// Mitsubishi GX Works2 project: BookEX6_49 PID   PLC: Q13UDV

// global labels: Global
VAR_GLOBAL
  bVar0 AT M5000 : BOOL;
  abArray0 AT M5010 : ARRAY [0..49] OF BOOL;
  sStr0 AT D5000 : STRING[199];
  sStr1 AT D5100 : STRING[199];
  sStr2 AT D5200 : STRING[199];
  sStr3 AT D5300 : STRING[199];
  sStr4 AT D5400 : STRING[199];
  sStr5 AT D5500 : STRING[199];
  sStr6 AT D5600 : STRING[199];
  sStr7 AT D5700 : STRING[199];
  sStr8 AT D5800 : STRING[199];
  sStr9 AT D5900 : STRING[199];
  iVar0 AT D4500 : INT;
  iVar1 AT D4501 : INT;
  iVar2 AT D4502 : INT;
  iVar3 AT D4503 : INT;
  iVar4 AT D4504 : INT;
  iVar5 AT D4505 : INT;
  iVar6 AT D4506 : INT;
  iVar7 AT D4507 : INT;
  iVar8 AT D4508 : INT;
  iVar9 AT D4509 : INT;
  dVar0 AT D4510 : DINT;
  dVar1 AT D4512 : DINT;
  dVar2 AT D4514 : DINT;
  dVar3 AT D4516 : DINT;
  dVar4 AT D4518 : DINT;
  dVar5 AT D4520 : DINT;
  dVar6 AT D4522 : DINT;
  dVar7 AT D4524 : DINT;
  dVar8 AT D4526 : DINT;
  dVar9 AT D4528 : DINT;
  wVar0 AT D4530 : WORD;
  wVar1 AT D4531 : WORD;
  wVar2 AT D4532 : WORD;
  wVar3 AT D4533 : WORD;
  wVar4 AT D4534 : WORD;
  wVar5 AT D4535 : WORD;
  wVar6 AT D4536 : WORD;
  wVar7 AT D4537 : WORD;
  wVar8 AT D4538 : WORD;
  wVar9 AT D4539 : WORD;
  dwVar0 AT D4540 : DWORD;
  dwVar1 AT D4542 : DWORD;
  dwVar2 AT D4544 : DWORD;
  dwVar3 AT D4546 : DWORD;
  dwVar4 AT D4548 : DWORD;
  dwVar5 AT D4550 : DWORD;
  dwVar6 AT D4552 : DWORD;
  dwVar7 AT D4554 : DWORD;
  dwVar8 AT D4556 : DWORD;
  dwVar9 AT D4558 : DWORD;
  fsVar0 AT D4560 : REAL;
  fsVar1 AT D4562 : REAL;
  fsVar2 AT D4564 : REAL;
  fsVar3 AT D4566 : REAL;
  fsVar4 AT D4568 : REAL;
  fsVar5 AT D4570 : REAL;
  fsVar6 AT D4572 : REAL;
  fsVar7 AT D4574 : REAL;
  fsVar8 AT D4576 : REAL;
  fsVar9 AT D4578 : REAL;
  fdVar0 AT D4580 : LREAL;
  tTime0 AT D4620 : TIME;
  tTime1 AT D4622 : TIME;
  tTime2 AT D4624 : TIME;
  tTime3 AT D4626 : TIME;
  tTime4 AT D4628 : TIME;
  tTime5 AT D4630 : TIME;
  tTime6 AT D4632 : TIME;
  tTime7 AT D4634 : TIME;
  tTime8 AT D4636 : TIME;
  tTime9 AT D4638 : TIME;
  tTime10 AT D4640 : TIME;
  bVar1 AT M5001 : BOOL;
  bVar2 AT M5002 : BOOL;
  bVar3 AT M5003 : BOOL;
  bVar4 AT M5004 : BOOL;
  bVar5 AT M5005 : BOOL;
  bVar6 AT M5006 : BOOL;
  bVar7 AT M5007 : BOOL;
  bVar8 AT M5008 : BOOL;
  bVar9 AT M5009 : BOOL;
  abArray1 AT M5060 : ARRAY [0..49] OF BOOL;
  abArray2 AT M5110 : ARRAY [0..49] OF BOOL;
  abArray3 AT M5160 : ARRAY [0..49] OF BOOL;
  abArray4 AT M5210 : ARRAY [0..49] OF BOOL;
  abArray5 AT M5260 : ARRAY [0..49] OF BOOL;
  abArray6 AT M5310 : ARRAY [0..49] OF BOOL;
  abArray7 AT M5360 : ARRAY [0..49] OF BOOL;
  abArray8 AT M5410 : ARRAY [0..49] OF BOOL;
  abArray9 AT M5460 : ARRAY [0..49] OF BOOL;
  fdVar1 AT D4584 : LREAL;
  fdVar2 AT D4588 : LREAL;
  fdVar3 AT D4592 : LREAL;
  fdVar4 AT D4596 : LREAL;
  fdVar5 AT D4600 : LREAL;
  fdVar6 AT D4604 : LREAL;
  fdVar7 AT D4608 : LREAL;
  fdVar8 AT D4612 : LREAL;
  fdVar9 AT D4616 : LREAL;
  afsPen0 AT D2000 : ARRAY [0..499] OF REAL;
  afsPen1 AT D3000 : ARRAY [0..499] OF REAL;
END_VAR
// user libraries (not included): HMI

PROGRAM ExPIDGraph
VAR
  ix : INT;
  iy : INT;
  fsPV : REAL;
  fsEV : REAL;
  fsLastEV : REAL;
  fsIV : REAL;
  fsDV : REAL;
  fsSV : REAL;
  fsKp : REAL;
  fsKi : REAL;
  fsKd : REAL;
  fsDT : REAL;
  fsOut : REAL;
  fsLastPV : REAL;
END_VAR
;
IF SM402 THEN
	fsVar8 := -20.0;		(* Min *)
	fsVar9 := 20.0;		(* Max *)
	ix := 0;
	fsSV := 10.0;
	fsPV := 0.0;
	fsIV := 0.0;
	fsDV := 0.0;
	fsLastEV := 0.0;
	fsVar0 := 2.0;
	fsVar1 := 10.0;
	fsVar2 := 0.2;
	FOR iy:=0 TO 359 DO 
		IF iy > 300 THEN
			afsPen0[iy] := 0.0;
		ELSIF iy > 170 THEN
			afsPen0[iy] := fsSV * -1.0;
		ELSIF iy > 40 THEN
			afsPen0[iy] := fsSV;
		ELSE
			afsPen0[iy] := 0.0;
		END_IF;
	END_FOR;		
	sStr0 := 'P Gain';
	sStr1 := 'I Gain';
	sStr2 := 'D Gain';
	sStr3 := '';
	sStr4 := '';
	fsVar3 := 0.0;
	iVar4 := 0;
END_IF;

IF LDP(TRUE, SM410)  THEN 
	CASE ix OF 
		0..359 : (* PID-Control *)
					fsDT := 0.1;			
					fsEV := fsPV - afsPen0[ix];
					fsIV := fsIV + fsEV * fsDT;
					fsDV := (fsEV - fsLastEV) / fsDT;
					fsLastEV := fsEV;  
					fsOut := fsVar0 * fsEV + fsVar1 * fsIV + fsVar2 * fsDV; 
					fsPV := fsLastPV - fsOut * fsDT;
					fsLastPV := fsPV;
					(* Limit *)
					IF (fsPV > fsVar9) THEN fsPV := fsVar9;  END_IF;
					IF (fsPV < fsVar8) THEN  fsPV := fsVar8;  END_IF;
 					FOR iy:=ix TO 359 DO 
						afsPen1[iy] := fsPV;
					END_FOR;    
					ix := ix + 1;		
	ELSE
		ix := 0;
		fsPV := 0.0;
		fsIV := 0.0;
		fsDV := 0.0;
		fsLastEV := 0.0;
		FOR iy:=0 TO 359 DO 
				afsPen1[iy] := 0.0;
		END_FOR;		
	END_CASE;
END_IF;
END_PROGRAM

PROGRAM ExPID
VAR
  Mov8INT_1 : Mov8INT;
  aCtrlData : ARRAY [0..28] OF INT;
  iSV : INT;
  iPV : INT;
  iMV : INT;
  Mov8INT_2 : Mov8INT;
  Mov8INT_3 : Mov8INT;
  fsMV : REAL;
  HMI06_1 : HMI06;
END_VAR
(* structured ladder/FBD written out as ST: instructions are called as NAME(EN, inputs, outputs); _pN, _eN, _tN stand for wires *)
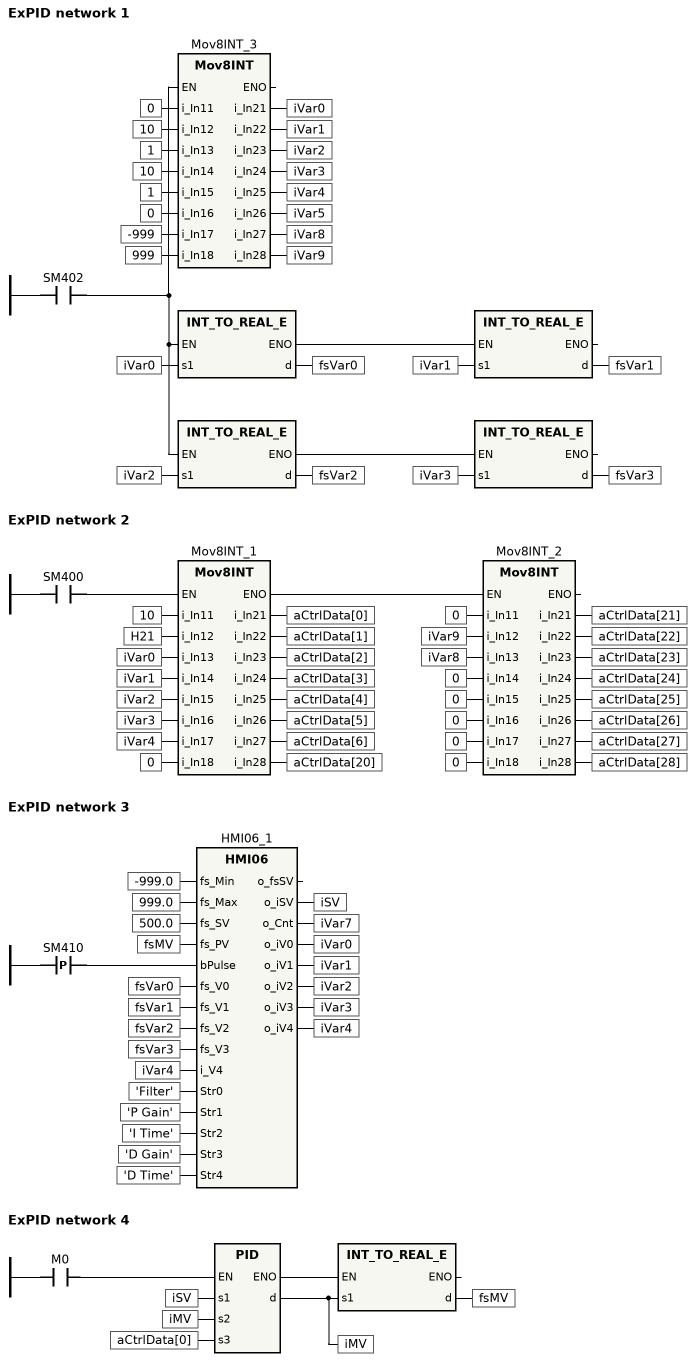
(* network 1 *)
Mov8INT_3(EN := SM402, i_In11 := 0, i_In12 := 10, i_In13 := 1, i_In14 := 10, i_In15 := 1, i_In16 := 0, i_In17 := -999, i_In18 := 999, i_In21 => iVar0, i_In22 => iVar1, i_In23 => iVar2, i_In24 => iVar3, i_In25 => iVar4, i_In26 => iVar5, i_In27 => iVar8, i_In28 => iVar9);
_e1 := INT_TO_REAL_E(SM402, iVar0, fsVar0);
INT_TO_REAL_E(_e1, iVar1, fsVar1);
_e2 := INT_TO_REAL_E(SM402, iVar2, fsVar2);
INT_TO_REAL_E(_e2, iVar3, fsVar3);
(* network 2 *)
Mov8INT_1(EN := SM400, i_In11 := 10, i_In12 := H21, i_In13 := iVar0, i_In14 := iVar1, i_In15 := iVar2, i_In16 := iVar3, i_In17 := iVar4, i_In18 := 0, i_In21 => aCtrlData[0], i_In22 => aCtrlData[1], i_In23 => aCtrlData[2], i_In24 => aCtrlData[3], i_In25 => aCtrlData[4], i_In26 => aCtrlData[5], i_In27 => aCtrlData[6], i_In28 => aCtrlData[20]);
Mov8INT_2(EN := Mov8INT_1.ENO, i_In11 := 0, i_In12 := iVar9, i_In13 := iVar8, i_In14 := 0, i_In15 := 0, i_In16 := 0, i_In17 := 0, i_In18 := 0, i_In21 => aCtrlData[21], i_In22 => aCtrlData[22], i_In23 => aCtrlData[23], i_In24 => aCtrlData[24], i_In25 => aCtrlData[25], i_In26 => aCtrlData[26], i_In27 => aCtrlData[27], i_In28 => aCtrlData[28]);
(* network 3 *)
HMI06_1(fs_Min := -999.0, fs_Max := 999.0, fs_SV := 500.0, fs_PV := fsMV, bPulse := LDP(TRUE, SM410), fs_V0 := fsVar0, fs_V1 := fsVar1, fs_V2 := fsVar2, fs_V3 := fsVar3, i_V4 := iVar4, Str0 := 'Filter', Str1 := 'P Gain', Str2 := 'I Time', Str3 := 'D Gain', Str4 := 'D Time', o_iSV => iSV, o_Cnt => iVar7, o_iV0 => iVar0, o_iV1 => iVar1, o_iV2 => iVar2, o_iV3 => iVar3, o_iV4 => iVar4);
(* network 4 *)
_e1 := PID(M0, iSV, iMV, aCtrlData[0], iMV);
INT_TO_REAL_E(_e1, iMV, fsMV);
END_PROGRAM

PROGRAM ExInexactPRMW
VAR
  Mov8INT_1 : Mov8INT;
  Mov8INT_2 : Mov8INT;
  aCtrlData : ARRAY [0..99] OF INT;
  aCtrlCont : ARRAY [0..172] OF INT;
  Mov4INT_1 : Mov4INT;
  HMI06_1 : HMI06;
  iMV : INT;
  fsMV : REAL;
  Mov8INT_3 : Mov8INT;
  fsSV : REAL;
  iSV : INT;
  Mov8INT_4 : Mov8INT;
  Mov8INT_5 : Mov8INT;
  Mov4INT_2 : Mov4INT;
  aPrmwData : ARRAY [0..99] OF INT;
END_VAR
(* structured ladder/FBD written out as ST: instructions are called as NAME(EN, inputs, outputs); _pN, _eN, _tN stand for wires *)
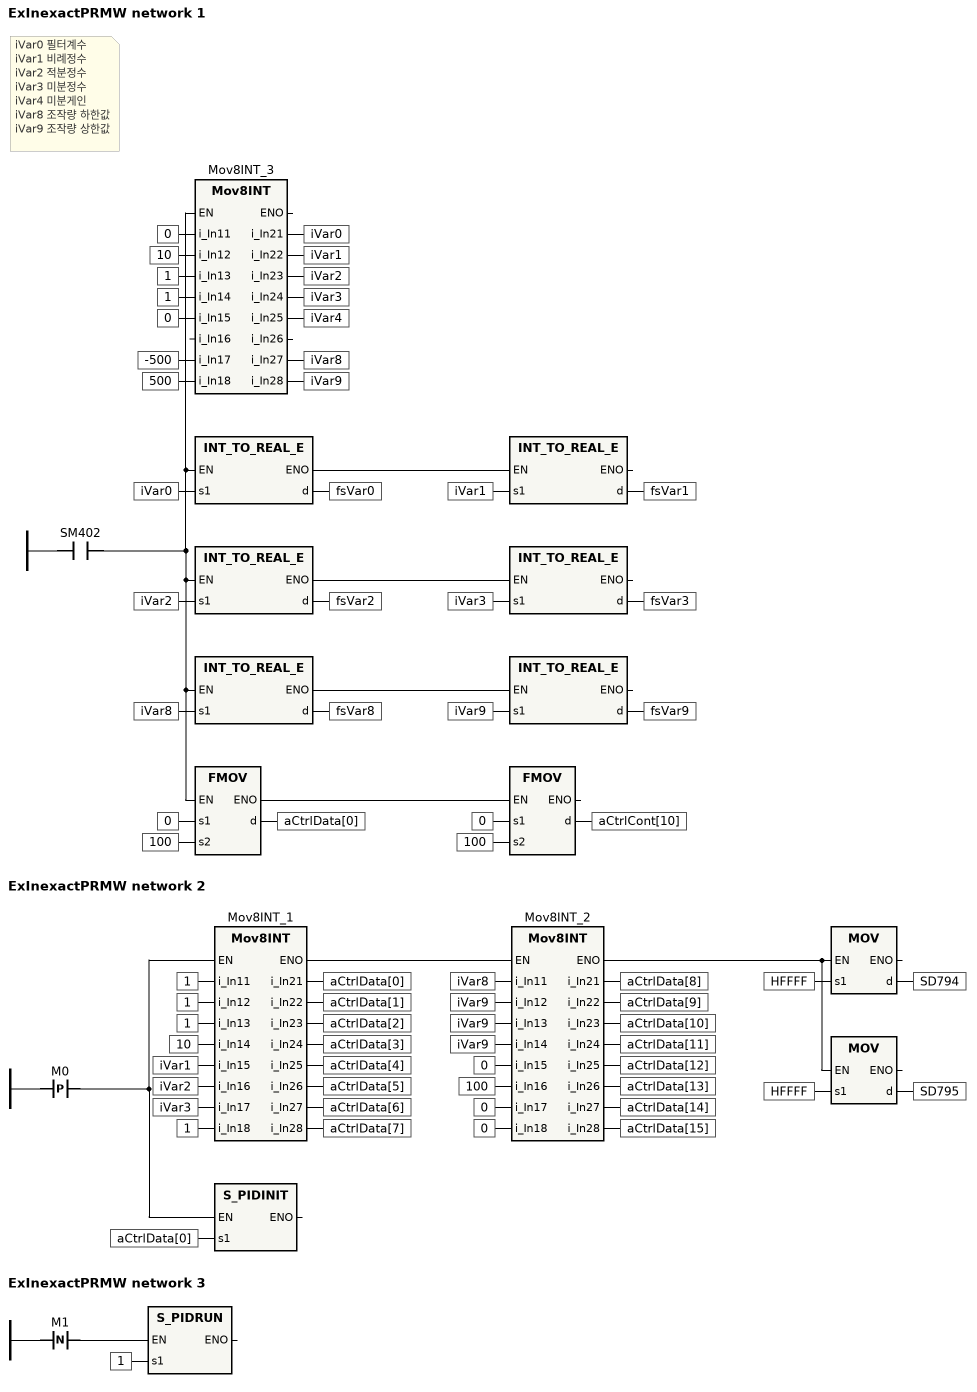
(* network 1 *)
(* iVar0 필터계수 / iVar1 비례정수 / iVar2 적분정수 / iVar3 미분정수 / iVar4 미분게인 / iVar8 조작량 하한값 / iVar9 조작량 상한값 *)
Mov8INT_3(EN := SM402, i_In11 := 0, i_In12 := 10, i_In13 := 1, i_In14 := 1, i_In15 := 0, i_In17 := -500, i_In18 := 500, i_In21 => iVar0, i_In22 => iVar1, i_In23 => iVar2, i_In24 => iVar3, i_In25 => iVar4, i_In27 => iVar8, i_In28 => iVar9);
_e1 := INT_TO_REAL_E(SM402, iVar0, fsVar0);
INT_TO_REAL_E(_e1, iVar1, fsVar1);
_e2 := INT_TO_REAL_E(SM402, iVar2, fsVar2);
INT_TO_REAL_E(_e2, iVar3, fsVar3);
_e3 := INT_TO_REAL_E(SM402, iVar8, fsVar8);
INT_TO_REAL_E(_e3, iVar9, fsVar9);
_e4 := FMOV(SM402, 0, 100, aCtrlData[0]);
FMOV(_e4, 0, 100, aCtrlCont[10]);
(* network 2 *)
_p1 := LDP(TRUE, M0);
Mov8INT_1(EN := _p1, i_In11 := 1, i_In12 := 1, i_In13 := 1, i_In14 := 10, i_In15 := iVar1, i_In16 := iVar2, i_In17 := iVar3, i_In18 := 1, i_In21 => aCtrlData[0], i_In22 => aCtrlData[1], i_In23 => aCtrlData[2], i_In24 => aCtrlData[3], i_In25 => aCtrlData[4], i_In26 => aCtrlData[5], i_In27 => aCtrlData[6], i_In28 => aCtrlData[7]);
Mov8INT_2(EN := Mov8INT_1.ENO, i_In11 := iVar8, i_In12 := iVar9, i_In13 := iVar9, i_In14 := iVar9, i_In15 := 0, i_In16 := 100, i_In17 := 0, i_In18 := 0, i_In21 => aCtrlData[8], i_In22 => aCtrlData[9], i_In23 => aCtrlData[10], i_In24 => aCtrlData[11], i_In25 => aCtrlData[12], i_In26 => aCtrlData[13], i_In27 => aCtrlData[14], i_In28 => aCtrlData[15]);
MOV(Mov8INT_2.ENO, HFFFF, SD794);
MOV(Mov8INT_2.ENO, HFFFF, SD795);
S_PIDINIT(_p1, aCtrlData[0]);
(* network 3 *)
S_PIDRUN(LDF(TRUE, M1), 1);
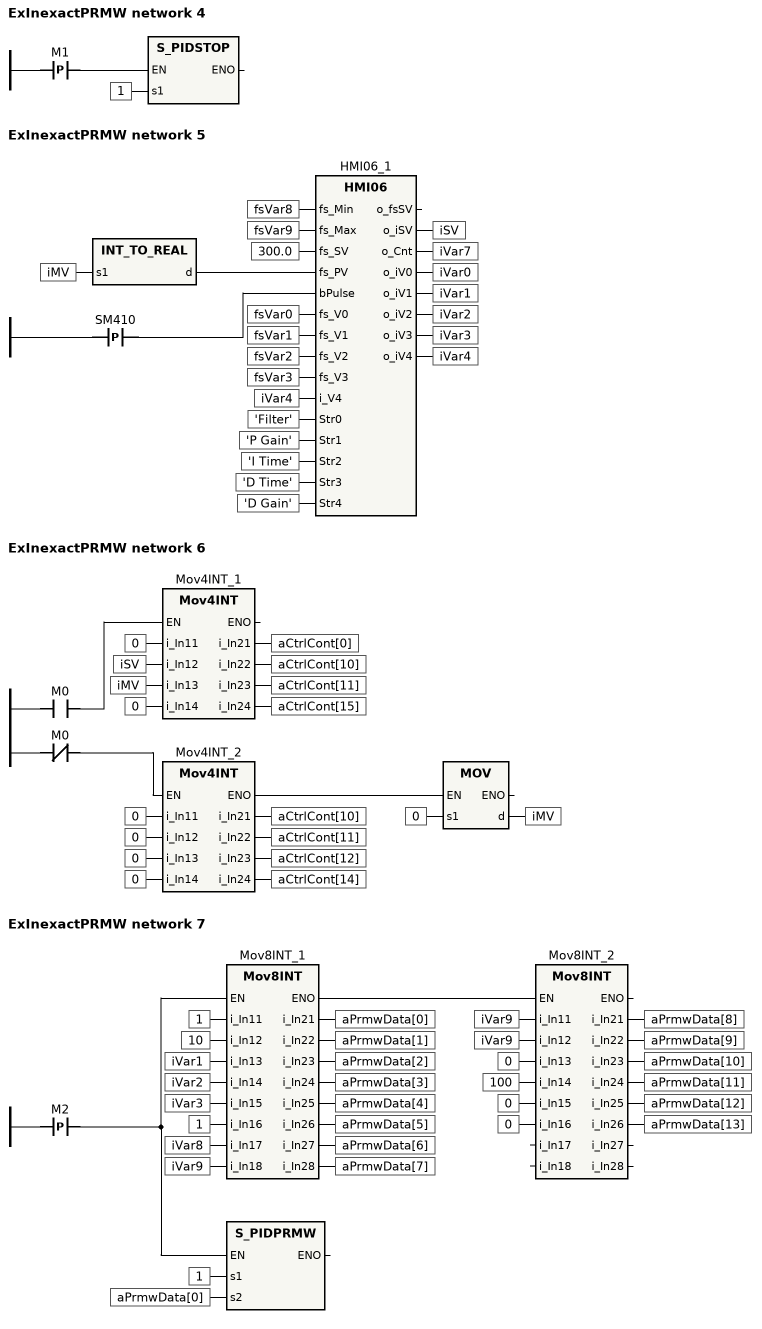
(* network 4 *)
S_PIDSTOP(LDP(TRUE, M1), 1);
(* network 5 *)
HMI06_1(fs_Min := fsVar8, fs_Max := fsVar9, fs_SV := 300.0, fs_PV := INT_TO_REAL(iMV), bPulse := LDP(TRUE, SM410), fs_V0 := fsVar0, fs_V1 := fsVar1, fs_V2 := fsVar2, fs_V3 := fsVar3, i_V4 := iVar4, Str0 := 'Filter', Str1 := 'P Gain', Str2 := 'I Time', Str3 := 'D Time', Str4 := 'D Gain', o_iSV => iSV, o_Cnt => iVar7, o_iV0 => iVar0, o_iV1 => iVar1, o_iV2 => iVar2, o_iV3 => iVar3, o_iV4 => iVar4);
(* network 6 *)
Mov4INT_1(EN := M0, i_In11 := 0, i_In12 := iSV, i_In13 := iMV, i_In14 := 0, i_In21 => aCtrlCont[0], i_In22 => aCtrlCont[10], i_In23 => aCtrlCont[11], i_In24 => aCtrlCont[15]);
Mov4INT_2(EN := NOT M0, i_In11 := 0, i_In12 := 0, i_In13 := 0, i_In14 := 0, i_In21 => aCtrlCont[10], i_In22 => aCtrlCont[11], i_In23 => aCtrlCont[12], i_In24 => aCtrlCont[14]);
MOV(Mov4INT_2.ENO, 0, iMV);
(* network 7 *)
_p1 := LDP(TRUE, M2);
Mov8INT_1(EN := _p1, i_In11 := 1, i_In12 := 10, i_In13 := iVar1, i_In14 := iVar2, i_In15 := iVar3, i_In16 := 1, i_In17 := iVar8, i_In18 := iVar9, i_In21 => aPrmwData[0], i_In22 => aPrmwData[1], i_In23 => aPrmwData[2], i_In24 => aPrmwData[3], i_In25 => aPrmwData[4], i_In26 => aPrmwData[5], i_In27 => aPrmwData[6], i_In28 => aPrmwData[7]);
Mov8INT_2(EN := Mov8INT_1.ENO, i_In11 := iVar9, i_In12 := iVar9, i_In13 := 0, i_In14 := 100, i_In15 := 0, i_In16 := 0, i_In21 => aPrmwData[8], i_In22 => aPrmwData[9], i_In23 => aPrmwData[10], i_In24 => aPrmwData[11], i_In25 => aPrmwData[12], i_In26 => aPrmwData[13]);
S_PIDPRMW(_p1, 1, aPrmwData[0]);
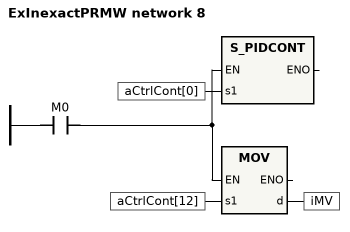
(* network 8 *)
S_PIDCONT(M0, aCtrlCont[0]);
MOV(M0, aCtrlCont[12], iMV);
END_PROGRAM

PROGRAM ExInexact
VAR
  Mov8INT_1 : Mov8INT;
  Mov8INT_2 : Mov8INT;
  aCtrlData : ARRAY [0..99] OF INT;
  aCtrlCont : ARRAY [0..172] OF INT;
  Mov4INT_1 : Mov4INT;
  HMI06_1 : HMI06;
  iMV : INT;
  fsMV : REAL;
  Mov8INT_3 : Mov8INT;
  fsSV : REAL;
  iSV : INT;
  Mov8INT_4 : Mov8INT;
  Mov8INT_5 : Mov8INT;
  Mov4INT_2 : Mov4INT;
END_VAR
(* structured ladder/FBD written out as ST: instructions are called as NAME(EN, inputs, outputs); _pN, _eN, _tN stand for wires *)
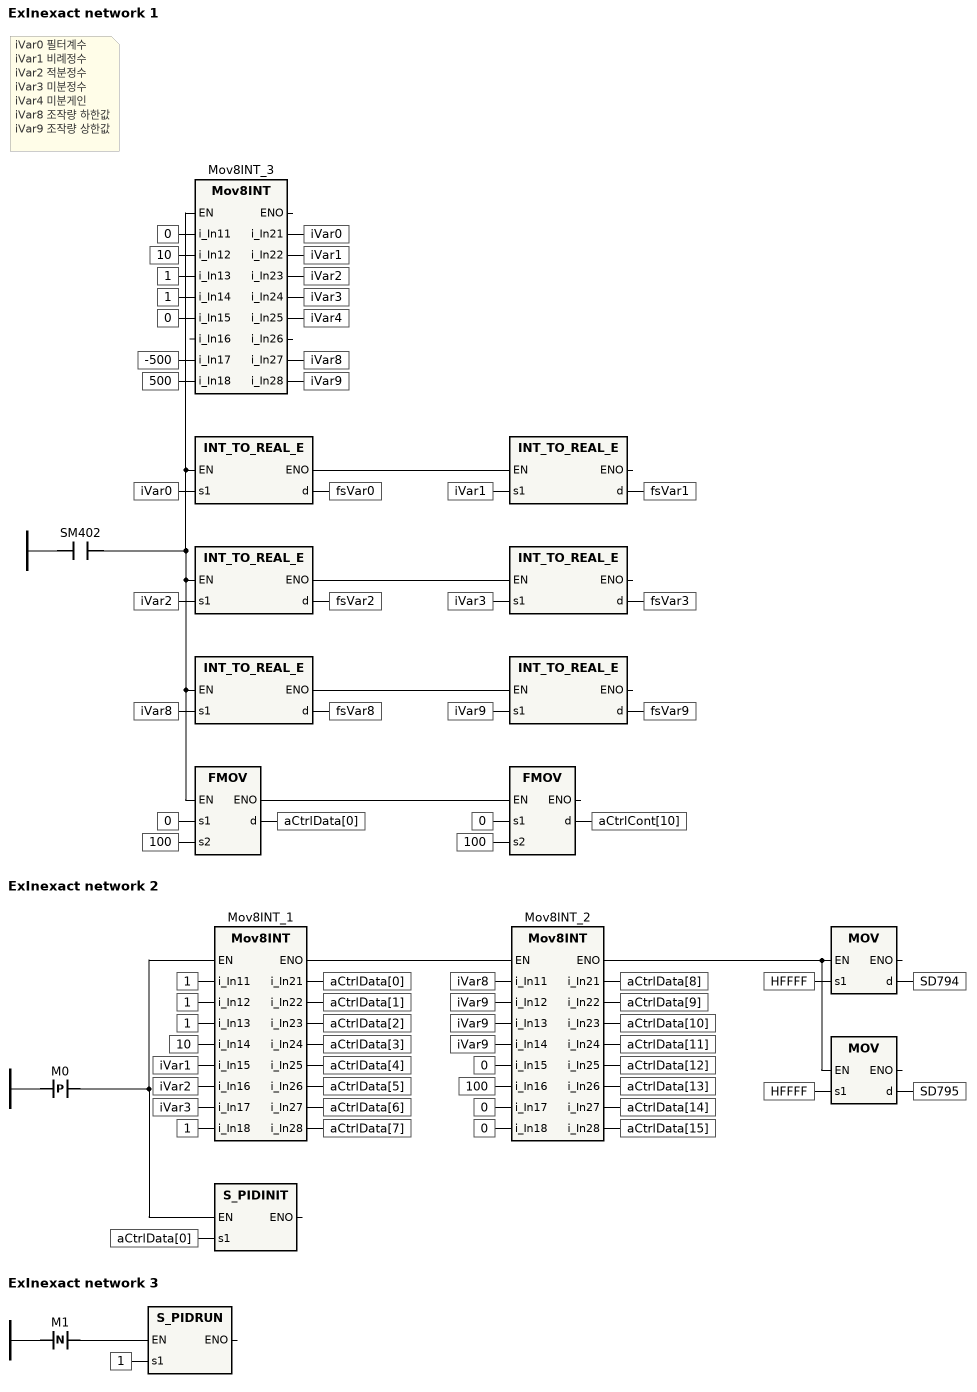
(* network 1 *)
(* iVar0 필터계수 / iVar1 비례정수 / iVar2 적분정수 / iVar3 미분정수 / iVar4 미분게인 / iVar8 조작량 하한값 / iVar9 조작량 상한값 *)
Mov8INT_3(EN := SM402, i_In11 := 0, i_In12 := 10, i_In13 := 1, i_In14 := 1, i_In15 := 0, i_In17 := -500, i_In18 := 500, i_In21 => iVar0, i_In22 => iVar1, i_In23 => iVar2, i_In24 => iVar3, i_In25 => iVar4, i_In27 => iVar8, i_In28 => iVar9);
_e1 := INT_TO_REAL_E(SM402, iVar0, fsVar0);
INT_TO_REAL_E(_e1, iVar1, fsVar1);
_e2 := INT_TO_REAL_E(SM402, iVar2, fsVar2);
INT_TO_REAL_E(_e2, iVar3, fsVar3);
_e3 := INT_TO_REAL_E(SM402, iVar8, fsVar8);
INT_TO_REAL_E(_e3, iVar9, fsVar9);
_e4 := FMOV(SM402, 0, 100, aCtrlData[0]);
FMOV(_e4, 0, 100, aCtrlCont[10]);
(* network 2 *)
_p1 := LDP(TRUE, M0);
Mov8INT_1(EN := _p1, i_In11 := 1, i_In12 := 1, i_In13 := 1, i_In14 := 10, i_In15 := iVar1, i_In16 := iVar2, i_In17 := iVar3, i_In18 := 1, i_In21 => aCtrlData[0], i_In22 => aCtrlData[1], i_In23 => aCtrlData[2], i_In24 => aCtrlData[3], i_In25 => aCtrlData[4], i_In26 => aCtrlData[5], i_In27 => aCtrlData[6], i_In28 => aCtrlData[7]);
Mov8INT_2(EN := Mov8INT_1.ENO, i_In11 := iVar8, i_In12 := iVar9, i_In13 := iVar9, i_In14 := iVar9, i_In15 := 0, i_In16 := 100, i_In17 := 0, i_In18 := 0, i_In21 => aCtrlData[8], i_In22 => aCtrlData[9], i_In23 => aCtrlData[10], i_In24 => aCtrlData[11], i_In25 => aCtrlData[12], i_In26 => aCtrlData[13], i_In27 => aCtrlData[14], i_In28 => aCtrlData[15]);
MOV(Mov8INT_2.ENO, HFFFF, SD794);
MOV(Mov8INT_2.ENO, HFFFF, SD795);
S_PIDINIT(_p1, aCtrlData[0]);
(* network 3 *)
S_PIDRUN(LDF(TRUE, M1), 1);
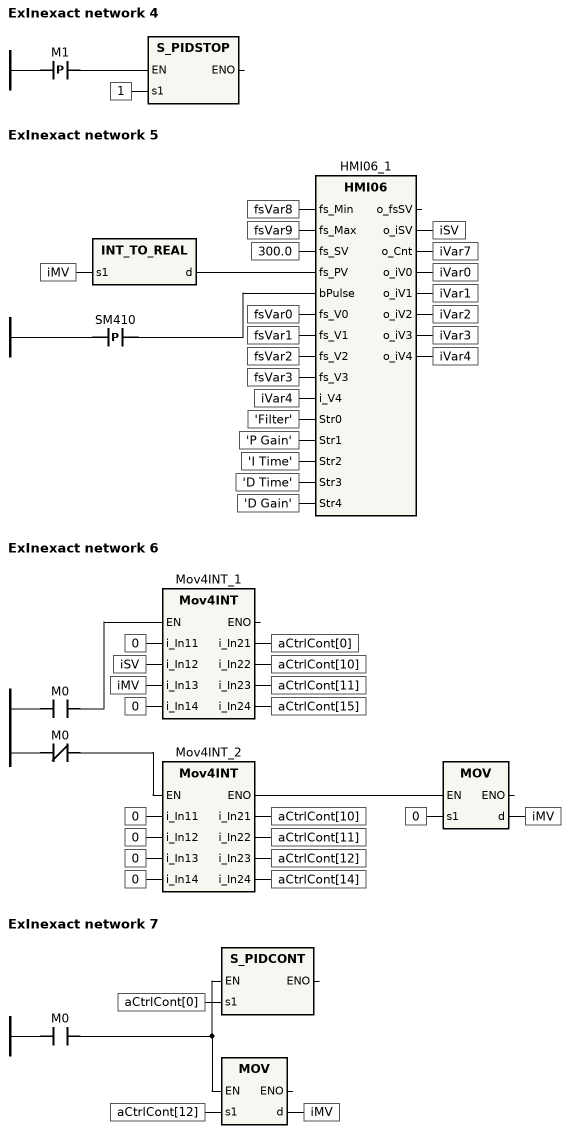
(* network 4 *)
S_PIDSTOP(LDP(TRUE, M1), 1);
(* network 5 *)
HMI06_1(fs_Min := fsVar8, fs_Max := fsVar9, fs_SV := 300.0, fs_PV := INT_TO_REAL(iMV), bPulse := LDP(TRUE, SM410), fs_V0 := fsVar0, fs_V1 := fsVar1, fs_V2 := fsVar2, fs_V3 := fsVar3, i_V4 := iVar4, Str0 := 'Filter', Str1 := 'P Gain', Str2 := 'I Time', Str3 := 'D Time', Str4 := 'D Gain', o_iSV => iSV, o_Cnt => iVar7, o_iV0 => iVar0, o_iV1 => iVar1, o_iV2 => iVar2, o_iV3 => iVar3, o_iV4 => iVar4);
(* network 6 *)
Mov4INT_1(EN := M0, i_In11 := 0, i_In12 := iSV, i_In13 := iMV, i_In14 := 0, i_In21 => aCtrlCont[0], i_In22 => aCtrlCont[10], i_In23 => aCtrlCont[11], i_In24 => aCtrlCont[15]);
Mov4INT_2(EN := NOT M0, i_In11 := 0, i_In12 := 0, i_In13 := 0, i_In14 := 0, i_In21 => aCtrlCont[10], i_In22 => aCtrlCont[11], i_In23 => aCtrlCont[12], i_In24 => aCtrlCont[14]);
MOV(Mov4INT_2.ENO, 0, iMV);
(* network 7 *)
S_PIDCONT(M0, aCtrlCont[0]);
MOV(M0, aCtrlCont[12], iMV);
END_PROGRAM

PROGRAM ExExact
VAR
  Mov8INT_1 : Mov8INT;
  Mov8INT_2 : Mov8INT;
  aCtrlData : ARRAY [0..99] OF INT;
  aCtrlCont : ARRAY [0..172] OF INT;
  Mov4INT_1 : Mov4INT;
  iMV : INT;
  fsMV : REAL;
  Mov8INT_3 : Mov8INT;
  fsSV : REAL;
  iSV : INT;
  Mov8INT_4 : Mov8INT;
  Mov8INT_5 : Mov8INT;
  Mov4INT_2 : Mov4INT;
  HMI06_1 : HMI06;
END_VAR
(* structured ladder/FBD written out as ST: instructions are called as NAME(EN, inputs, outputs); _pN, _eN, _tN stand for wires *)
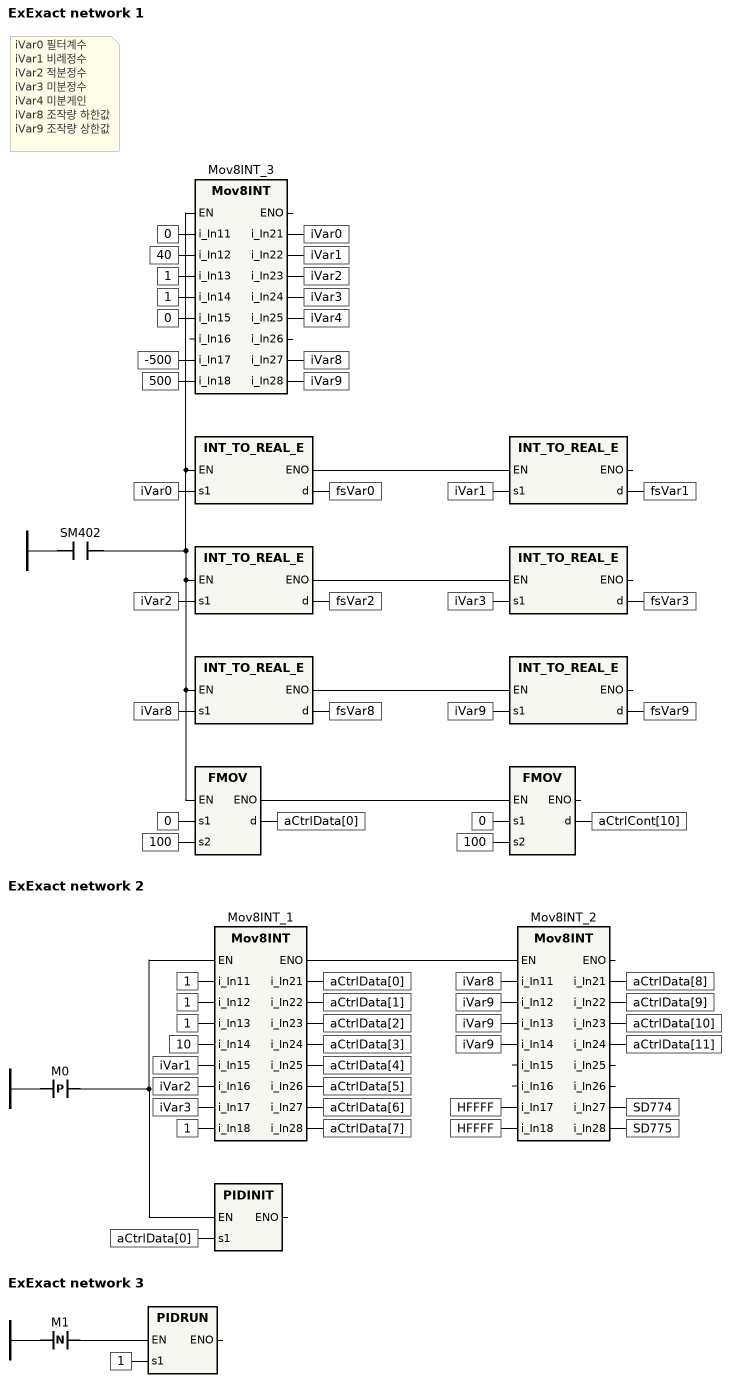
(* network 1 *)
(* iVar0 필터계수 / iVar1 비례정수 / iVar2 적분정수 / iVar3 미분정수 / iVar4 미분게인 / iVar8 조작량 하한값 / iVar9 조작량 상한값 *)
Mov8INT_3(EN := SM402, i_In11 := 0, i_In12 := 40, i_In13 := 1, i_In14 := 1, i_In15 := 0, i_In17 := -500, i_In18 := 500, i_In21 => iVar0, i_In22 => iVar1, i_In23 => iVar2, i_In24 => iVar3, i_In25 => iVar4, i_In27 => iVar8, i_In28 => iVar9);
_e1 := INT_TO_REAL_E(SM402, iVar0, fsVar0);
INT_TO_REAL_E(_e1, iVar1, fsVar1);
_e2 := INT_TO_REAL_E(SM402, iVar2, fsVar2);
INT_TO_REAL_E(_e2, iVar3, fsVar3);
_e3 := INT_TO_REAL_E(SM402, iVar8, fsVar8);
INT_TO_REAL_E(_e3, iVar9, fsVar9);
_e4 := FMOV(SM402, 0, 100, aCtrlData[0]);
FMOV(_e4, 0, 100, aCtrlCont[10]);
(* network 2 *)
_p1 := LDP(TRUE, M0);
Mov8INT_1(EN := _p1, i_In11 := 1, i_In12 := 1, i_In13 := 1, i_In14 := 10, i_In15 := iVar1, i_In16 := iVar2, i_In17 := iVar3, i_In18 := 1, i_In21 => aCtrlData[0], i_In22 => aCtrlData[1], i_In23 => aCtrlData[2], i_In24 => aCtrlData[3], i_In25 => aCtrlData[4], i_In26 => aCtrlData[5], i_In27 => aCtrlData[6], i_In28 => aCtrlData[7]);
Mov8INT_2(EN := Mov8INT_1.ENO, i_In11 := iVar8, i_In12 := iVar9, i_In13 := iVar9, i_In14 := iVar9, i_In17 := HFFFF, i_In18 := HFFFF, i_In21 => aCtrlData[8], i_In22 => aCtrlData[9], i_In23 => aCtrlData[10], i_In24 => aCtrlData[11], i_In27 => SD774, i_In28 => SD775);
PIDINIT(_p1, aCtrlData[0]);
(* network 3 *)
PIDRUN(LDF(TRUE, M1), 1);
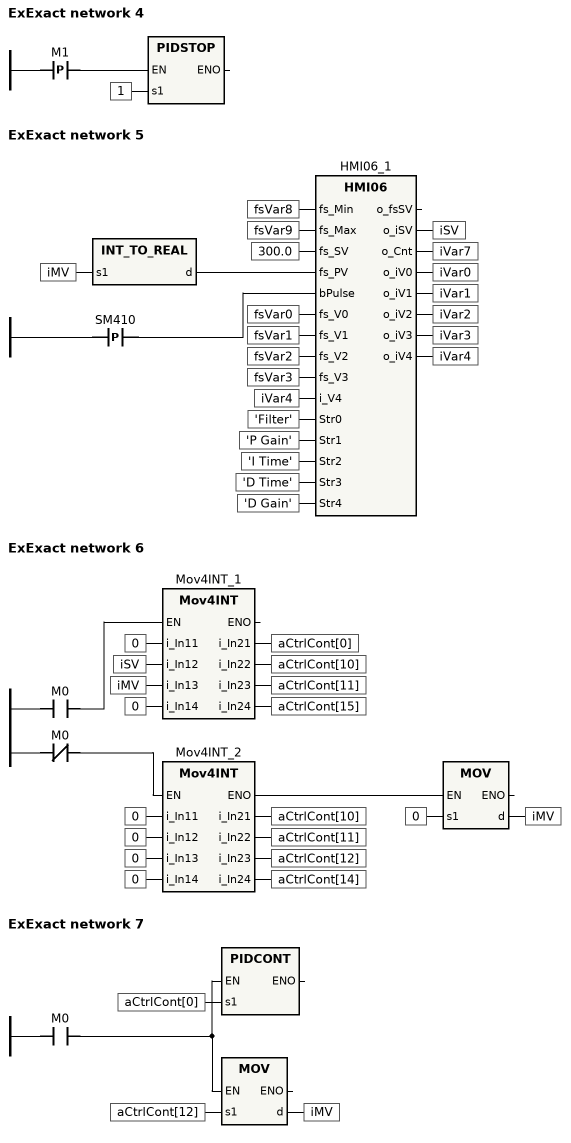
(* network 4 *)
PIDSTOP(LDP(TRUE, M1), 1);
(* network 5 *)
HMI06_1(fs_Min := fsVar8, fs_Max := fsVar9, fs_SV := 300.0, fs_PV := INT_TO_REAL(iMV), bPulse := LDP(TRUE, SM410), fs_V0 := fsVar0, fs_V1 := fsVar1, fs_V2 := fsVar2, fs_V3 := fsVar3, i_V4 := iVar4, Str0 := 'Filter', Str1 := 'P Gain', Str2 := 'I Time', Str3 := 'D Time', Str4 := 'D Gain', o_iSV => iSV, o_Cnt => iVar7, o_iV0 => iVar0, o_iV1 => iVar1, o_iV2 => iVar2, o_iV3 => iVar3, o_iV4 => iVar4);
(* network 6 *)
Mov4INT_1(EN := M0, i_In11 := 0, i_In12 := iSV, i_In13 := iMV, i_In14 := 0, i_In21 => aCtrlCont[0], i_In22 => aCtrlCont[10], i_In23 => aCtrlCont[11], i_In24 => aCtrlCont[15]);
Mov4INT_2(EN := NOT M0, i_In11 := 0, i_In12 := 0, i_In13 := 0, i_In14 := 0, i_In21 => aCtrlCont[10], i_In22 => aCtrlCont[11], i_In23 => aCtrlCont[12], i_In24 => aCtrlCont[14]);
MOV(Mov4INT_2.ENO, 0, iMV);
(* network 7 *)
PIDCONT(M0, aCtrlCont[0]);
MOV(M0, aCtrlCont[12], iMV);
END_PROGRAM

PROGRAM ExExactPRMW
VAR
  Mov8INT_1 : Mov8INT;
  Mov8INT_2 : Mov8INT;
  aCtrlData : ARRAY [0..99] OF INT;
  aCtrlCont : ARRAY [0..172] OF INT;
  Mov4INT_1 : Mov4INT;
  HMI06_1 : HMI06;
  iMV : INT;
  fsMV : REAL;
  Mov8INT_3 : Mov8INT;
  fsSV : REAL;
  iSV : INT;
  Mov8INT_4 : Mov8INT;
  Mov8INT_5 : Mov8INT;
  Mov4INT_2 : Mov4INT;
  aPrmwData : ARRAY [0..99] OF INT;
END_VAR
(* structured ladder/FBD written out as ST: instructions are called as NAME(EN, inputs, outputs); _pN, _eN, _tN stand for wires *)
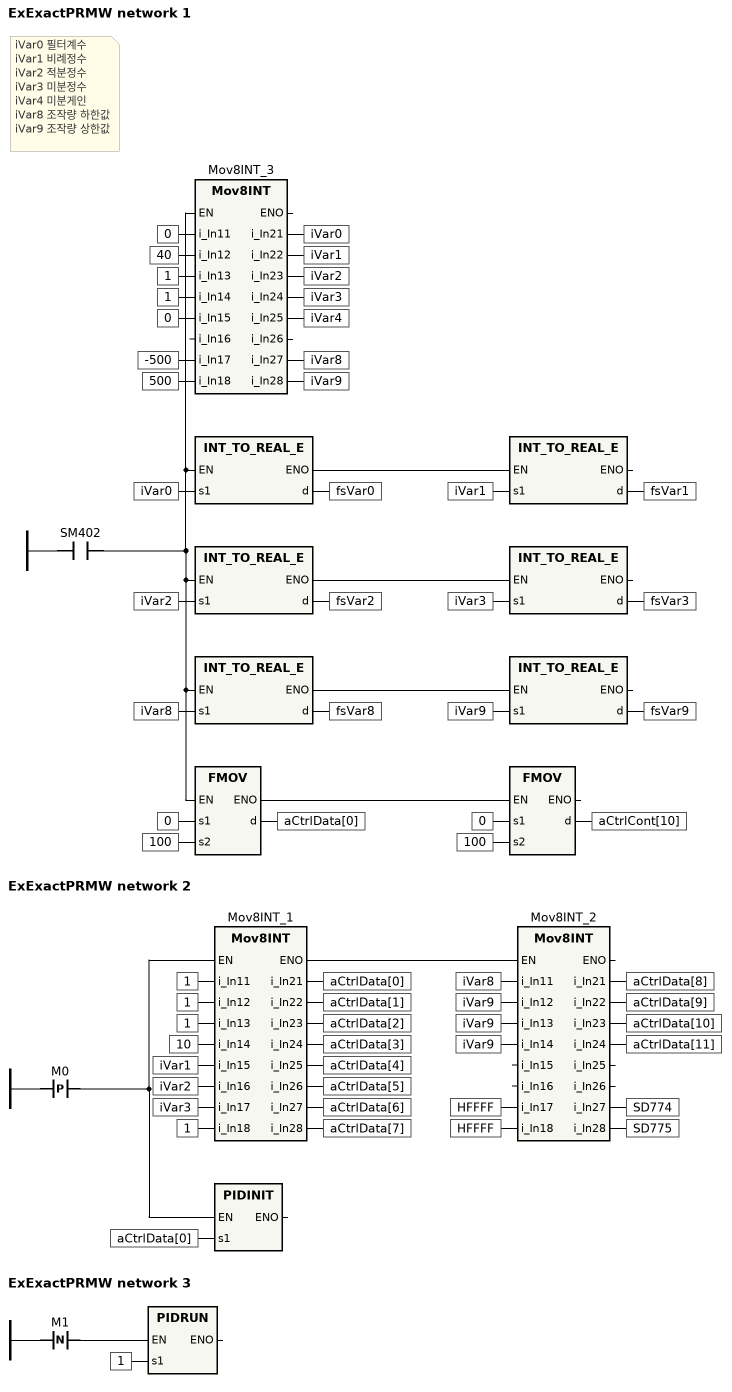
(* network 1 *)
(* iVar0 필터계수 / iVar1 비례정수 / iVar2 적분정수 / iVar3 미분정수 / iVar4 미분게인 / iVar8 조작량 하한값 / iVar9 조작량 상한값 *)
Mov8INT_3(EN := SM402, i_In11 := 0, i_In12 := 40, i_In13 := 1, i_In14 := 1, i_In15 := 0, i_In17 := -500, i_In18 := 500, i_In21 => iVar0, i_In22 => iVar1, i_In23 => iVar2, i_In24 => iVar3, i_In25 => iVar4, i_In27 => iVar8, i_In28 => iVar9);
_e1 := INT_TO_REAL_E(SM402, iVar0, fsVar0);
INT_TO_REAL_E(_e1, iVar1, fsVar1);
_e2 := INT_TO_REAL_E(SM402, iVar2, fsVar2);
INT_TO_REAL_E(_e2, iVar3, fsVar3);
_e3 := INT_TO_REAL_E(SM402, iVar8, fsVar8);
INT_TO_REAL_E(_e3, iVar9, fsVar9);
_e4 := FMOV(SM402, 0, 100, aCtrlData[0]);
FMOV(_e4, 0, 100, aCtrlCont[10]);
(* network 2 *)
_p1 := LDP(TRUE, M0);
Mov8INT_1(EN := _p1, i_In11 := 1, i_In12 := 1, i_In13 := 1, i_In14 := 10, i_In15 := iVar1, i_In16 := iVar2, i_In17 := iVar3, i_In18 := 1, i_In21 => aCtrlData[0], i_In22 => aCtrlData[1], i_In23 => aCtrlData[2], i_In24 => aCtrlData[3], i_In25 => aCtrlData[4], i_In26 => aCtrlData[5], i_In27 => aCtrlData[6], i_In28 => aCtrlData[7]);
Mov8INT_2(EN := Mov8INT_1.ENO, i_In11 := iVar8, i_In12 := iVar9, i_In13 := iVar9, i_In14 := iVar9, i_In17 := HFFFF, i_In18 := HFFFF, i_In21 => aCtrlData[8], i_In22 => aCtrlData[9], i_In23 => aCtrlData[10], i_In24 => aCtrlData[11], i_In27 => SD774, i_In28 => SD775);
PIDINIT(_p1, aCtrlData[0]);
(* network 3 *)
PIDRUN(LDF(TRUE, M1), 1);
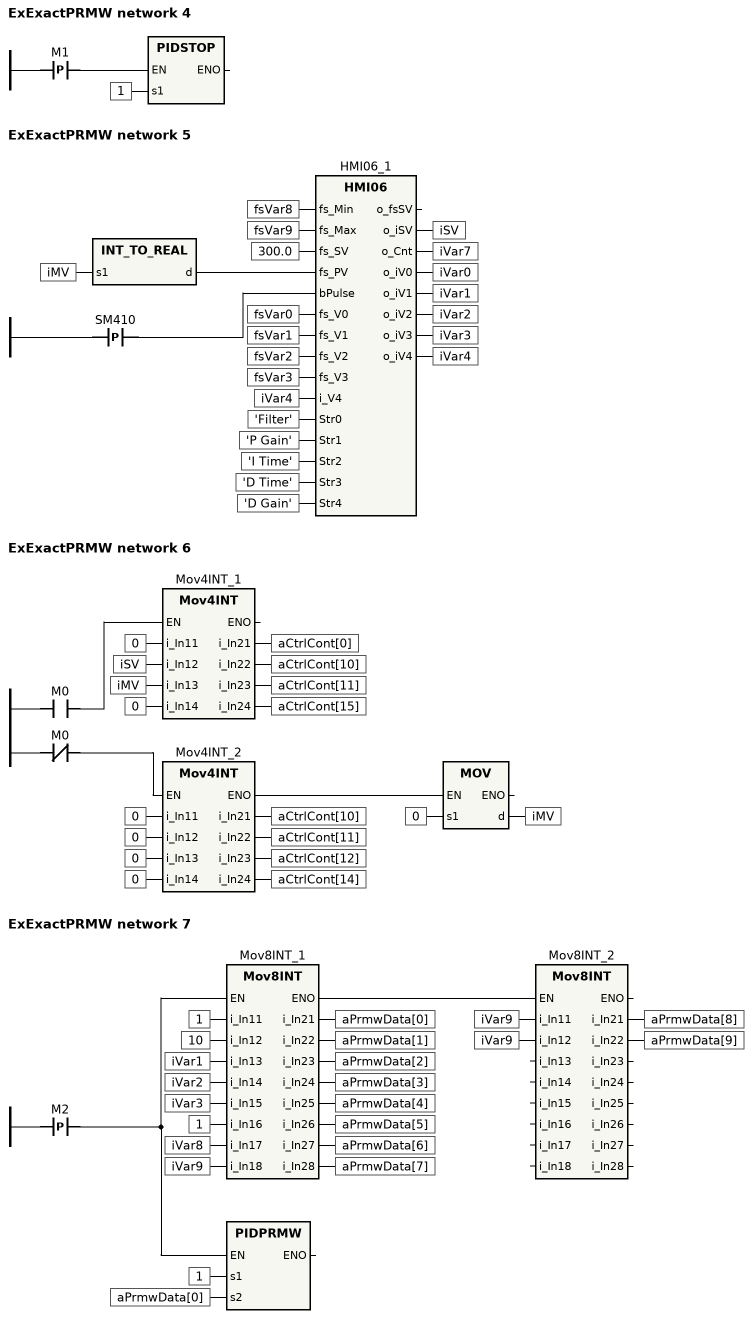
(* network 4 *)
PIDSTOP(LDP(TRUE, M1), 1);
(* network 5 *)
HMI06_1(fs_Min := fsVar8, fs_Max := fsVar9, fs_SV := 300.0, fs_PV := INT_TO_REAL(iMV), bPulse := LDP(TRUE, SM410), fs_V0 := fsVar0, fs_V1 := fsVar1, fs_V2 := fsVar2, fs_V3 := fsVar3, i_V4 := iVar4, Str0 := 'Filter', Str1 := 'P Gain', Str2 := 'I Time', Str3 := 'D Time', Str4 := 'D Gain', o_iSV => iSV, o_Cnt => iVar7, o_iV0 => iVar0, o_iV1 => iVar1, o_iV2 => iVar2, o_iV3 => iVar3, o_iV4 => iVar4);
(* network 6 *)
Mov4INT_1(EN := M0, i_In11 := 0, i_In12 := iSV, i_In13 := iMV, i_In14 := 0, i_In21 => aCtrlCont[0], i_In22 => aCtrlCont[10], i_In23 => aCtrlCont[11], i_In24 => aCtrlCont[15]);
Mov4INT_2(EN := NOT M0, i_In11 := 0, i_In12 := 0, i_In13 := 0, i_In14 := 0, i_In21 => aCtrlCont[10], i_In22 => aCtrlCont[11], i_In23 => aCtrlCont[12], i_In24 => aCtrlCont[14]);
MOV(Mov4INT_2.ENO, 0, iMV);
(* network 7 *)
_p1 := LDP(TRUE, M2);
Mov8INT_1(EN := _p1, i_In11 := 1, i_In12 := 10, i_In13 := iVar1, i_In14 := iVar2, i_In15 := iVar3, i_In16 := 1, i_In17 := iVar8, i_In18 := iVar9, i_In21 => aPrmwData[0], i_In22 => aPrmwData[1], i_In23 => aPrmwData[2], i_In24 => aPrmwData[3], i_In25 => aPrmwData[4], i_In26 => aPrmwData[5], i_In27 => aPrmwData[6], i_In28 => aPrmwData[7]);
Mov8INT_2(EN := Mov8INT_1.ENO, i_In11 := iVar9, i_In12 := iVar9, i_In21 => aPrmwData[8], i_In22 => aPrmwData[9]);
PIDPRMW(_p1, 1, aPrmwData[0]);
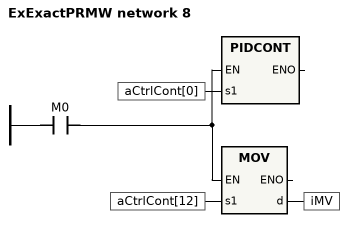
(* network 8 *)
PIDCONT(M0, aCtrlCont[0]);
MOV(M0, aCtrlCont[12], iMV);
END_PROGRAM
